(* IEC 61131-3 sources: RL_MAR/experiments/comparison/llm4plc/results/gpt-4o_20260507_114630/20260507_121818, 1 file *)

(* ---- generated_code_iteration_0.st ---- *)
plaintext
START_ST
FUNCTION_BLOCK PetFeederControl
VAR_INPUT
    CurrentTime : TIME; (* Current system time input *)
END_VAR
VAR_OUTPUT
    FoodDispense : BOOL; (* Food dispenser control signal *)
END_VAR
VAR
    (* Feeding time constants *)
    FeedTime1 : TIME := T#8H0M0S; (* First feeding time - 8:00 AM *)
    FeedTime2 : TIME := T#12H0M0S; (* Second feeding time - 12:00 PM *)
    FeedTime3 : TIME := T#18H0M0S; (* Third feeding time - 6:00 PM *)

    (* Internal state variables *)
    state : INT := 0; (* Current state of the system *)
    prevState : INT := 0; (* Previous state of the system, optional for debugging *)

    (* Food amount variable (currently unused) *)
    FoodAmount : INT := 50; (* Amount of food to dispense in grams *)
END_VAR

(* State Machine Logic *)
IF state = 0 THEN
    (* STATE 0: IDLE *)
    FoodDispense := FALSE;

    (* Transition to STATE 1: Dispensing for FeedTime1 *)
    IF (CurrentTime >= FeedTime1) AND (CurrentTime < FeedTime1 + T#30S) THEN
        state := 1;
    END_IF

    (* Transition to STATE 2: Dispensing for FeedTime2 *)
    IF (CurrentTime >= FeedTime2) AND (CurrentTime < FeedTime2 + T#30S) THEN
        state := 2;
    END_IF

    (* Transition to STATE 3: Dispensing for FeedTime3 *)
    IF (CurrentTime >= FeedTime3) AND (CurrentTime < FeedTime3 + T#30S) THEN
        state := 3;
    END_IF

ELSIF state = 1 THEN
    (* STATE 1: DISPENSING FOOD FOR FEEDTIME1 *)
    FoodDispense := TRUE;

    (* Transition back to STATE 0: IDLE after 30 seconds *)
    IF CurrentTime >= FeedTime1 + T#30S THEN
        state := 0;
    END_IF

ELSIF state = 2 THEN
    (* STATE 2: DISPENSING FOOD FOR FEEDTIME2 *)
    FoodDispense := TRUE;

    (* Transition back to STATE 0: IDLE after 30 seconds *)
    IF CurrentTime >= FeedTime2 + T#30S THEN
        state := 0;
    END_IF

ELSIF state = 3 THEN
    (* STATE 3: DISPENSING FOOD FOR FEEDTIME3 *)
    FoodDispense := TRUE;

    (* Transition back to STATE 0: IDLE after 30 seconds *)
    IF CurrentTime >= FeedTime3 + T#30S THEN
        state := 0;
    END_IF
END_IF

(* Optional: Store the previous state for debugging or tracking *)
prevState := state;

END_FUNCTION_BLOCK
END_ST
